    SpotL L0216190191BP20\VFO:=210,vSpot,nomtcp2\WObj:=BS_1606_1A;
    SpotL L0216190193BP20\VFO:=210,vSpot,nomtcp2\WObj:=BS_1606_1A;
    SpotL L0216190195BP20\VFO:=210\Vorhub_Auf,vSpot,nomtcp2\WObj:=BS_1606_1A;

    SpotL G0216190269BP20\VFO:=210,vSpot,nomtcp2\WObj:=BS_1606_1A;

    SpotL G0216190139BP20\VFO:=210,vSpot,nomtcp2\WObj:=BS_1606_1A;
    SpotL G0216190137BP20\VFO:=210,vSpot,nomtcp2\WObj:=BS_1606_1A;

    MoveJ LHP_110,vSchnell,z100,nomtcp2\WObj:=BS_1606_1A;
    SpotL G0216190143BP20\VFO:=210,vSpot,nomtcp2\WObj:=BS_1606_1A;
    SpotL G0216190753BP20\VFO:=210,vSpot,nomtcp2\WObj:=BS_1606_1A;
    SpotL G0216190751BP20\VFO:=210,vSpot,nomtcp2\WObj:=BS_1606_1A;

    SpotL G0216190187BP20\VFO:=210,vSpot,nomtcp2\WObj:=BS_1606_1A;
    SpotL G0216190185BP20\VFO:=210,vSpot,nomtcp2\WObj:=BS_1606_1A;
    SpotL G0216190183BP20\VFO:=210,vSpot,nomtcp2\WObj:=BS_1606_1A;
    SpotL G0216190181BP20\VFO:=210,vSpot,nomtcp2\WObj:=BS_1606_1A;
    SpotL G0216190179BP20\VFO:=210,vSpot,nomtcp2\WObj:=BS_1606_1A;
    SpotL G0216190177BP20\VFO:=210\Vorhub_Auf,vSpot,nomtcp2\WObj:=BS_1606_1A;

    MoveJ LHP_115,vSchnell,z100,nomtcp2\WObj:=BS_1606_1A;
    MoveJ LHP_120,vSchnell,z100,nomtcp2\WObj:=BS_1606_1A;
    MoveJ LHP_125,vSchnell,z100,nomtcp2\WObj:=BS_1606_1A;

    SpotL G0216190175BP20\VFO:=210,vSpot,nomtcp2\WObj:=BS_1606_1A;
    SpotL G0216190173BP20\VFO:=210\Vorhub_Auf,vSpot,nomtcp2\WObj:=BS_1606_1A;


    MoveJ LHP_130,vSchnell,z100,nomtcp2\WObj:=BS_1606_1A;
    MoveJ LHP_135,vSchnell,z100,nomtcp2\WObj:=BS_1606_1A;


    MoveJ LHP_155,vSchnell,z100,nomtcp2\WObj:=BS_1606_1A;

    MoveJ LHP_160,vSchnell,fine,nomtcp2\WObj:=BS_1606_1A;

    SpotL G0216190221BP20\VFO:=210\Vorhub_Auf,vSpot,nomtcp2\WObj:=BS_1606_1A;

    MoveJ LHP_165,vSchnell,fine,nomtcp2\WObj:=BS_1606_1A;

    MoveJ LHP_170,vSchnell,z100,nomtcp2\WObj:=BS_1606_1A;
    MoveJ LHP_175,vSchnell,z100,nomtcp2\WObj:=BS_1606_1A;
    MoveJ LHP_180,vSchnell,z100,nomtcp2\WObj:=BS_1606_1A;
    SpotL G0216190213BP20\VFO:=210\Vorhub_Auf,vSpot,nomtcp2\WObj:=BS_1606_1A;

    SpotL G0216190225BP20\VFO:=210,vSpot,nomtcp2\WObj:=BS_1606_1A;

    KOLLISION_ZONE 5\Freigabe;

    KOLLISION_ZONE 6\Freigabe;

    SpotL G0216190223BP20\VFO:=210,vSpot,nomtcp2\WObj:=BS_1606_1A;
    SpotL G0216190415BP20\VFO:=210\Vorhub_Auf,vSpot,nomtcp2\WObj:=BS_1606_1A;

    MoveJ LHP_185,vSchnell,z100,nomtcp2\WObj:=BS_1606_1A;
    MoveJ LHP_190,vSchnell,z100,nomtcp2\WObj:=BS_1606_1A;

    MoveJ LHP_195,vSchnell,fine,nomtcp2\WObj:=BS_1606_1A;

    ABL 254\ABL_SET;

    MoveJ LHP_200,vSchnell,z50,nomtcp2\WObj:=BS_1606_1A;
    MoveJ LHP_205,vSchnell,z100,nomtcp2\WObj:=BS_1606_1A;

    MoveJ ToolHome2,vSchnell,fine,nomtcp2;

    MoveJ ToolHome2,vSchnell,fine,nomtcp2;

    ABL 254\ABL_WAIT;

    ABL 255\ABL_SET;
  ENDPROC
  PROC swp_223300_0_st1606_2_copy()
    CONST robtarget LHP_000:=[[-343.969,-1509.453,-77.326],[0.6961739,0.14374174,0.69977224,-0.07070346],[0,1,-2,1],[9E9,9E9,9E9,9E9,9E9,9E9]];
    CONST robtarget LHP_005:=[[299.16,-1077.798,-195.105],[0.81965727,0.1372977,0.5457811,0.10693151],[0,1,-2,1],[9E9,9E9,9E9,9E9,9E9,9E9]];
    CONST robtarget LHP_010:=[[459.824,-945.357,-253.673],[0.83997643,0.0634096,0.49949673,0.20229144],[0,1,-2,1],[9E9,9E9,9E9,9E9,9E9,9E9]];
    CONST robtarget LHP_015:=[[429.2348,-845.8104,-123.9084],[0.77240807,0.12149542,0.5837386,0.21880084],[-1,1,-2,1],[9E9,9E9,9E9,9E9,9E9,9E9]];
    CONST robtarget LHP_020:=[[320.538,-988.972,23.814],[0.6084938,0.46778333,0.6390498,-0.05029308],[-1,1,-2,1],[9E9,9E9,9E9,9E9,9E9,9E9]];
    CONST robtarget LHP_025:=[[168.143,-1310.857,-178.565],[0.08599422,0.69841975,0.30285692,-0.6427227],[-1,2,-1,1],[9E9,9E9,9E9,9E9,9E9,9E9]];
    CONST robtarget LHP_030:=[[380.362,-1002.808,-83.829],[0.25333694,-0.7020941,-0.251623,0.6160926],[-1,2,-1,1],[9E9,9E9,9E9,9E9,9E9,9E9]];
    CONST robtarget LHP_035:=[[387.125,-886.744,-129.57],[0.2696306,-0.7098945,-0.24714555,0.6018872],[-1,1,-1,1],[9E9,9E9,9E9,9E9,9E9,9E9]];
    CONST robtarget LHP_040:=[[387.123,-886.744,-129.569],[0.2696306,-0.7098945,-0.24714555,0.6018872],[-1,1,-1,1],[9E9,9E9,9E9,9E9,9E9,9E9]];
    CONST robtarget LHP_045:=[[380.362,-1002.808,-83.829],[0.25333694,-0.7020941,-0.251623,0.6160926],[-1,2,-1,1],[9E9,9E9,9E9,9E9,9E9,9E9]];
    CONST robtarget LHP_050:=[[554.345,-1088.494,69.835],[0.24868385,-0.69330287,-0.186217,0.65023893],[-1,2,-1,1],[9E9,9E9,9E9,9E9,9E9,9E9]];
    CONST robtarget LHP_055:=[[1180.85,-956.12,360.53],[0.26714,-0.700539,-0.204389,0.62937],[-1,2,-1,1],[9E+09,9E+09,9E+09,9E+09,9E+09,9E+09]];
    CONST robtarget LHP_060:=[[1158.045,-818.462,292.246],[0.1861414,-0.6960594,-0.18546282,0.6681738],[-1,2,-1,1],[9E9,9E9,9E9,9E9,9E9,9E9]];
    CONST robtarget LHP_065:=[[1158.052,-818.462,292.251],[0.18614723,-0.696061,-0.18545675,0.6681722],[-1,2,-1,1],[9E9,9E9,9E9,9E9,9E9,9E9]];
    CONST robtarget LHP_070:=[[1155.504,-852.264,349.625],[0.18613547,-0.6960606,-0.18545689,0.6681759],[-1,2,-1,1],[9E9,9E9,9E9,9E9,9E9,9E9]];
    CONST robtarget LHP_075:=[[1177.941,-956.109,360.508],[0.2671498,-0.70053387,-0.20438649,0.62937224],[-1,2,-1,1],[9E9,9E9,9E9,9E9,9E9,9E9]];
    CONST robtarget LHP_080:=[[1230.988,-1024.279,150.53],[0.4850452,-0.59317434,-0.34627607,0.54126537],[-1,3,-2,1],[9E9,9E9,9E9,9E9,9E9,9E9]];
    CONST robtarget LHP_085:=[[1153.64,-804.49,-163.93],[0.369472,-0.630736,-0.314437,0.605633],[-1,3,-2,1],[9E+09,9E+09,9E+09,9E+09,9E+09,9E+09]];
    CONST robtarget LHP_090:=[[1155.58,-802.37,-202.14],[0.378085,-0.6383,-0.289331,0.604907],[-1,3,-2,1],[9E+09,9E+09,9E+09,9E+09,9E+09,9E+09]];
    CONST robtarget LHP_095:=[[1160.786,-932.752,-118.293],[0.35632858,-0.6342394,-0.31263465,0.61076176],[-1,2,-2,1],[9E9,9E9,9E9,9E9,9E9,9E9]];
    CONST robtarget LHP_100:=[[1177.199138001,-1034.633545366,-134.68460502],[0.599530277,0.416484833,0.54592798,0.411176936],[-1,3,0,1],[9E9,9E9,9E9,9E9,9E9,9E9]];
    CONST robtarget LHP_105:=[[1261.553,-949.259,-168.645],[0.49878648,0.46502888,0.53270465,0.5011845],[-1,3,0,1],[9E9,9E9,9E9,9E9,9E9,9E9]];
    CONST robtarget LHP_110:=[[1293.638,-800.057,-53.414],[0.4487649,0.511483,0.47262233,0.5600208],[-1,3,0,1],[9E9,9E9,9E9,9E9,9E9,9E9]];
    CONST robtarget LHP_115:=[[1292.46,-1068.67,105.62],[0.537954,0.460499,0.543891,0.450254],[-1,3,0,1],[9E+09,9E+09,9E+09,9E+09,9E+09,9E+09]];
    CONST robtarget LHP_120:=[[1272.09,-1035.73,404.02],[0.665811,0.311525,0.616981,0.281039],[-1,2,1,1],[9E+09,9E+09,9E+09,9E+09,9E+09,9E+09]];
    CONST robtarget LHP_125:=[[1288.49,-827.17,318.14],[0.65686,0.248853,0.659538,0.267614],[-1,2,1,1],[9E+09,9E+09,9E+09,9E+09,9E+09,9E+09]];
    CONST robtarget LHP_130:=[[1282.834,-831.497,331.588],[0.6238299,0.28569758,0.64522505,0.3360026],[-1,2,1,1],[9E9,9E9,9E9,9E9,9E9,9E9]];
    CONST robtarget LHP_135:=[[1272.23,-1035.576,350.423],[0.6007957,0.3326514,0.61991906,0.3795892],[-1,2,0,1],[9E9,9E9,9E9,9E9,9E9,9E9]];
    CONST robtarget LHP_140:=[[1515.36,-1930.427,-710.889],[0.68370384,-0.3828575,0.5419457,0.30375],[-1,1,0,1],[9E9,9E9,9E9,9E9,9E9,9E9]];
    CONST robtarget LHP_145:=[[1508.39,-1126.698,-345.994],[0.7746838,-0.06633059,0.21093813,0.59242755],[-1,1,1,0],[9E9,9E9,9E9,9E9,9E9,9E9]];
    CONST robtarget LHP_150:=[[1193.732,-854.946,-340.29],[0.6808548,-0.006798419,0.021675188,0.7320661],[-1,1,0,0],[9E9,9E9,9E9,9E9,9E9,9E9]];
    CONST robtarget LHP_155:=[[1264.265,-860.681,-343.292],[0.6861445,-0.00817846,0.022382554,0.72707486],[-1,1,0,0],[9E9,9E9,9E9,9E9,9E9,9E9]];
    CONST robtarget LHP_160:=[[1378.915,-949.1688,-235.1],[0.7417187,-0.022747554,0.038135264,0.6692396],[-1,1,0,0],[9E9,9E9,9E9,9E9,9E9,9E9]];
    CONST robtarget LHP_165:=[[1378.916,-949.17,-239.0872],[0.7417192,-0.022746855,0.038135428,0.66923904],[-1,1,0,0],[9E9,9E9,9E9,9E9,9E9,9E9]];
    CONST robtarget LHP_170:=[[1378.918,-949.169,-333.471],[0.7417194,-0.0227467,0.038134836,0.6692388],[-1,1,0,0],[9E9,9E9,9E9,9E9,9E9,9E9]];
    CONST robtarget LHP_175:=[[1974.39,-993.49,-251.01],[0.870007,0.0142221,0.00384455,0.492819],[-1,1,0,0],[9E+09,9E+09,9E+09,9E+09,9E+09,9E+09]];
    CONST robtarget LHP_180:=[[1974.26,-983.70,-299.04],[0.00154131,-0.870074,-0.492907,-0.00333926],[-1,1,-2,0],[9E+09,9E+09,9E+09,9E+09,9E+09,9E+09]];
    CONST robtarget LHP_185:=[[2116.328,-924.396,-299.018],[0.023842378,-0.8889618,-0.4568781,-0.020995617],[-1,1,-2,0],[9E9,9E9,9E9,9E9,9E9,9E9]];
    CONST robtarget LHP_190:=[[1442.08,-914.903,-300.663],[0.022750434,-0.803067,-0.5947096,-0.029769931],[-1,1,-2,0],[9E9,9E9,9E9,9E9,9E9,9E9]];
    CONST robtarget LHP_195:=[[1433.186,-924.788,-304.288],[0.023560839,-0.8018969,-0.59623784,-0.030111516],[-1,1,-2,0],[9E9,9E9,9E9,9E9,9E9,9E9]];
    CONST robtarget LHP_200:=[[1929.389,-1029.042,-272.149],[0.16453815,0.87018114,0.45821258,-0.07585006],[-1,1,-2,0],[9E9,9E9,9E9,9E9,9E9,9E9]];
    CONST robtarget LHP_205:=[[1580.139,-1754.999,-225.61],[0.74780244,0.48078176,0.4354385,-0.14154042],[-1,1,-2,1],[9E9,9E9,9E9,9E9,9E9,9E9]];
    ! ------------------------------------------------------------
    ! Unterprogramm:
    ! Stand
    ! Daimler AG - Werk Ludwigsfelde
    ! ------------------------------------------------------------
    ! ************************************************************
    ! Kommentar: Achtung
    !            automatisch generiert!!!!!!!!!!!!!!!!!!
    ! ************************************************************

    ! Robotername:             1606R05
    ! Anlagenbezeichn:        Linie 16          Stations-Nr:  1606
    ! Stand / Version:        05.08.2009 / 1.1
    ! Name Bearbeiter:        Karmann
    ! Applikationssteuerung:  Punktschweissen
    ! Baumuster:              FHL T2 R2
    !
    !duplikat swp225500_0_st1606_2 kolision sind geendert

    INIT_SW_BASE;

    wkz_2_aufnehmen;

    MoveJ ToolHome2,vSchnell,fine,nomtcp2;
    !
    Vorhub\auf;
    !
    !KOLLISION_ZONE 9\Anfrage;
    KOLLISION_ZONE 5\Anfrage;
    !KOLLISION_ZONE 5\Freigabe;
    !
    MoveJ LHP_000,vSchnell,z100,nomtcp2\WObj:=BS_1606_1A;

    MoveJ LHP_005,vSchnell,z100,nomtcp2\WObj:=BS_1606_1A;
    MoveJ LHP_010,vSchnell,z100,nomtcp2\WObj:=BS_1606_1A;

    SpotL G0216001589BP20\VFO:=210,vSpot,nomtcp2\WObj:=BS_1606_1A;

    MoveL LHP_015,vSchnell,z100,nomtcp2\WObj:=BS_1606_1A;

    SpotL G0216001591BP20\VFO:=210,vSpot,nomtcp2\WObj:=BS_1606_1A;
    SpotL G0216001593BP20\VFO:=210,vSpot,nomtcp2\WObj:=BS_1606_1A;
    SpotL G0216001595BP20\VFO:=210,vSpot,nomtcp2\WObj:=BS_1606_1A;
    SpotL G0216001597BP20\VFO:=210,vSpot,nomtcp2\WObj:=BS_1606_1A;
    SpotL G0216001599BP20\VFO:=210,vSpot,nomtcp2\WObj:=BS_1606_1A;
    SpotL G0216001601BP20\VFO:=210\Vorhub_Auf,vSpot,nomtcp2\WObj:=BS_1606_1A;

    MoveJ LHP_020,vSchnell,z100,nomtcp2\WObj:=BS_1606_1A;
    MoveJ LHP_025,vSchnell,z100,nomtcp2\WObj:=BS_1606_1A;
    MoveJ LHP_030,vSchnell,z100,nomtcp2\WObj:=BS_1606_1A;
    MoveJ LHP_035,vSchnell,z100,nomtcp2\WObj:=BS_1606_1A;

    SpotL L0216047039BP20\VFO:=210\Vorhub_Auf,vSpot,nomtcp2\WObj:=BS_1606_1A;
    !
    KOLLISION_ZONE 9\Anfrage;
    !


    MoveJ LHP_040,vSchnell,z100,nomtcp2\WObj:=BS_1606_1A;
    MoveJ LHP_045,vSchnell,z100,nomtcp2\WObj:=BS_1606_1A;
    MoveJ LHP_050,vSchnell,z100,nomtcp2\WObj:=BS_1606_1A;
    MoveJ LHP_055,vSchnell,z100,nomtcp2\WObj:=BS_1606_1A;

    SpotL L0216190163BP20\VFO:=210,vSpot,nomtcp2\WObj:=BS_1606_1A;

    MoveL LHP_060,vSchnell,z100,nomtcp2\WObj:=BS_1606_1A;

    SpotL G0216190161BP20\VFO:=210\Vorhub_Auf,vSpot,nomtcp2\WObj:=BS_1606_1A;

    MoveJ LHP_065,vSchnell,z100,nomtcp2\WObj:=BS_1606_1A;
    MoveJ LHP_070,vSchnell,z100,nomtcp2\WObj:=BS_1606_1A;
    MoveJ LHP_075,vSchnell,z100,nomtcp2\WObj:=BS_1606_1A;
    MoveJ LHP_080,vSchnell,z100,nomtcp2\WObj:=BS_1606_1A;

    SpotL G0216190159BP20\VFO:=210,vSpot,nomtcp2\WObj:=BS_1606_1A;
    SpotL G0216190157BP20\VFO:=210,vSpot,nomtcp2\WObj:=BS_1606_1A;
    SpotL G0216190155BP20\VFO:=210,vSpot,nomtcp2\WObj:=BS_1606_1A;
    SpotL G0216190153BP20\VFO:=210,vSpot,nomtcp2\WObj:=BS_1606_1A;
    SpotL G0216190151BP20\VFO:=210,vSpot,nomtcp2\WObj:=BS_1606_1A;
    SpotL G0216190149BP20\VFO:=210,vSpot,nomtcp2\WObj:=BS_1606_1A;
    SpotL G0216190141BP20\VFO:=210,vSpot,nomtcp2\WObj:=BS_1606_1A;
    SpotL G0216190135BP20\VFO:=210,vSpot,nomtcp2\WObj:=BS_1606_1A;
    SpotL G0216190133BP20\VFO:=210,vSpot,nomtcp2\WObj:=BS_1606_1A;

    MoveJ LHP_085,vSchnell,z100,nomtcp2\WObj:=BS_1606_1A;
    MoveJ LHP_090,vSchnell,z100,nomtcp2\WObj:=BS_1606_1A;

    SpotL G0216190125BP20\VFO:=210\Vorhub_Auf,vSpot,nomtcp2\WObj:=BS_1606_1A;

    KOLLISION_ZONE 6\Anfrage;

    MoveJ LHP_095,vSchnell,z100,nomtcp2\WObj:=BS_1606_1A;
    MoveJ LHP_100,vSchnell,z100,nomtcp2\WObj:=BS_1606_1A;
    MoveJ LHP_105,vSchnell,z100,nomtcp2\WObj:=BS_1606_1A;

    !WaitUntil FALSE;
    !wstawic G0216190269BP20, zamiast G0216190127BP20
    SpotL G0216190269BP20\VFO:=210,vSpot,nomtcp2\WObj:=BS_1606_1A;

    !SpotL G0216190127BP20\VFO:=210,vSpot,nomtcp2\WObj:=BS_1606_1A;
    SpotL G0216190139BP20\VFO:=210,vSpot,nomtcp2\WObj:=BS_1606_1A;
    SpotL G0216190137BP20\VFO:=210,vSpot,nomtcp2\WObj:=BS_1606_1A;
    SpotL G0216190753BP20\VFO:=210,vSpot,nomtcp2\WObj:=BS_1606_1A;
    SpotL G0216190751BP20\VFO:=210,vSpot,nomtcp2\WObj:=BS_1606_1A;

    MoveJ LHP_110,vSchnell,z100,nomtcp2\WObj:=BS_1606_1A;

    SpotL G0216190143BP20\VFO:=210,vSpot,nomtcp2\WObj:=BS_1606_1A;
    SpotL G0216190187BP20\VFO:=210,vSpot,nomtcp2\WObj:=BS_1606_1A;
    SpotL G0216190185BP20\VFO:=210,vSpot,nomtcp2\WObj:=BS_1606_1A;
    SpotL G0216190183BP20\VFO:=210,vSpot,nomtcp2\WObj:=BS_1606_1A;
    SpotL G0216190181BP20\VFO:=210,vSpot,nomtcp2\WObj:=BS_1606_1A;
    SpotL G0216190179BP20\VFO:=210,vSpot,nomtcp2\WObj:=BS_1606_1A;
    SpotL G0216190177BP20\VFO:=210\Vorhub_Auf,vSpot,nomtcp2\WObj:=BS_1606_1A;

    MoveJ LHP_115,vSchnell,z100,nomtcp2\WObj:=BS_1606_1A;
    MoveJ LHP_120,vSchnell,z100,nomtcp2\WObj:=BS_1606_1A;
    MoveJ LHP_125,vSchnell,z100,nomtcp2\WObj:=BS_1606_1A;

    SpotL G0216190175BP20\VFO:=210,vSpot,nomtcp2\WObj:=BS_1606_1A;
    SpotL G0216190173BP20\VFO:=210\Vorhub_Auf,vSpot,nomtcp2\WObj:=BS_1606_1A;
    !
    KOLLISION_ZONE 1\Anfrage;

    MoveJ LHP_130,vSchnell,z100,nomtcp2\WObj:=BS_1606_1A;
    MoveJ LHP_135,vSchnell,z100,nomtcp2\WObj:=BS_1606_1A;
    MoveJ LHP_140,vSchnell,z100,nomtcp2\WObj:=BS_1606_1A;
    MoveJ LHP_145,vSchnell,z100,nomtcp2\WObj:=BS_1606_1A;
    MoveJ LHP_150,vSchnell,z100,nomtcp2\WObj:=BS_1606_1A;

    SpotL L0216190191BP20\VFO:=210,vSpot,nomtcp2\WObj:=BS_1606_1A;
    SpotL L0216190193BP20\VFO:=210,vSpot,nomtcp2\WObj:=BS_1606_1A;
    SpotL L0216190195BP20\VFO:=210\Vorhub_Auf,vSpot,nomtcp2\WObj:=BS_1606_1A;

    MoveJ LHP_155,vSchnell,z100,nomtcp2\WObj:=BS_1606_1A;

    MoveJ LHP_160,vSchnell,fine,nomtcp2\WObj:=BS_1606_1A;

    SpotL G0216190221BP20\VFO:=210\Vorhub_Auf,vSpot,nomtcp2\WObj:=BS_1606_1A;

    MoveJ LHP_165,vSchnell,fine,nomtcp2\WObj:=BS_1606_1A;

    MoveJ LHP_170,vSchnell,z100,nomtcp2\WObj:=BS_1606_1A;
    MoveJ LHP_175,vSchnell,z100,nomtcp2\WObj:=BS_1606_1A;
    MoveJ LHP_180,vSchnell,z100,nomtcp2\WObj:=BS_1606_1A;

    SpotL G0216190225BP20\VFO:=210,vSpot,nomtcp2\WObj:=BS_1606_1A;
    SpotL G0216190223BP20\VFO:=210,vSpot,nomtcp2\WObj:=BS_1606_1A;
    SpotL G0216190415BP20\VFO:=210\Vorhub_Auf,vSpot,nomtcp2\WObj:=BS_1606_1A;

    MoveJ LHP_185,vSchnell,z100,nomtcp2\WObj:=BS_1606_1A;
    MoveJ LHP_190,vSchnell,z100,nomtcp2\WObj:=BS_1606_1A;

    SpotL G0216190213BP20\VFO:=210\Vorhub_Auf,vSpot,nomtcp2\WObj:=BS_1606_1A;

    MoveJ LHP_195,vSchnell,fine,nomtcp2\WObj:=BS_1606_1A;

    ABL 254\ABL_SET;

    MoveJ LHP_200,vSchnell,z50,nomtcp2\WObj:=BS_1606_1A;
    MoveJ LHP_205,vSchnell,z100,nomtcp2\WObj:=BS_1606_1A;

    MoveJ ToolHome2,vSchnell,fine,nomtcp2;
    !
    KOLLISION_ZONE 1\Freigabe;
    !
    KOLLISION_ZONE 5\Freigabe;

    KOLLISION_ZONE 6\Freigabe;

    KOLLISION_ZONE 9\Freigabe;

    MoveJ ToolHome2,vSchnell,fine,nomtcp2;

    ABL 254\ABL_WAIT;

    ABL 255\ABL_SET;
  ENDPROC

ENDMODULE
